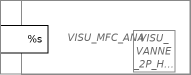
VISUALIZATION VISU_LIGNE_GAZ_ANA  // 191x75
VAR_IN_OUT
	m_Input_MACHINE:	BLOCK_MODE_MARCHE_V2_0;
	m_Input_MASSFLOW:	BLOCK_MFC_ANA2;
	m_Input_LIGNE_GAZ:	BLOCK_LIGNE_GAZ;		
END_VAR
    Frame (21,0 170x75)
        shows VISU_MFC_ANA(m_Input_MACHINE := m_Input_MACHINE, m_Input_MASSFLOW := m_Input_MASSFLOW, m_Input_LIGNE_GAZ := m_Input_LIGNE_GAZ)
    Frame (133,30 42x42)
        shows VISU_VANNE_2P_H_ACT2(m_Input_VANNE := m_Input_LIGNE_GAZ.VGI)
    Rectangle (0,25 48x28), "%s", text variable: m_Input_MASSFLOW.CONF_Util_Name
END_VISUALIZATION

(* stored: Version 1.1.0.1, ProductVersion 3.1.4024.10
   Visu VISU_LIGNE_GAZ_ANA: Id {55b347ed-ab48-446f-ba01-2ef91cc773f8} *)
